{attribute 'qualified_only'}
{attribute 'strict'}
{attribute 'to_string'}
TYPE E_BYTE :
(
	eMIN := 0,
	eVAL1,
	eVAL2,
	eVAL3,
	eMAX := 255
) BYTE;
END_TYPE

(* stored: Version 1.1.0.1
   DUT E_BYTE: Id {485092af-8816-4c74-a842-587770aad252} *)
